(* LS Electric XG5000 project: 20230520_Problems *)
(* PLC LSPLC *)

PROGRAM NewProgram (* task: 스캔 프로그램 *)
VAR
    P1 : BOOL;
    P10 : BOOL;
    P11 : BOOL;
    P2 : BOOL;
    P3 : BOOL;
END_VAR
VAR
    _e1 : R_TRIG;
END_VAR

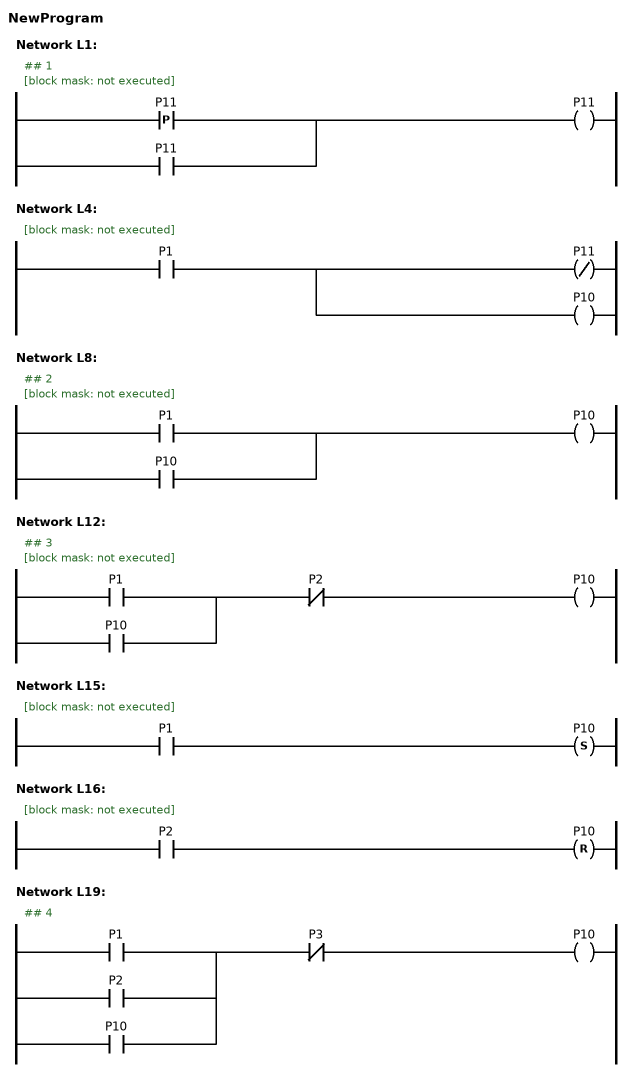
(* ## 1 *)
(* Rung L1 is block-masked: not executed *)
// _e1(CLK := P11);
// P11 := _e1.Q OR P11;
(* Rung L4 is block-masked: not executed *)
// P11 := NOT P1;
// P10 := P1;
(* ## 2 *)
(* Rung L8 is block-masked: not executed *)
// P10 := P1 OR P10;
(* ## 3 *)
(* Rung L12 is block-masked: not executed *)
// P10 := (P1 OR P10) AND NOT P2;
(* Rung L15 is block-masked: not executed *)
// IF P1 THEN P10 := TRUE; END_IF;
(* Rung L16 is block-masked: not executed *)
// IF P2 THEN P10 := FALSE; END_IF;
(* ## 4 *)
(* Rung L19 *)
P10 := (P1 OR P2 OR P10) AND NOT P3;
END_PROGRAM